(* IEC 61131-3 sources: programs/VI-54/VI-54_20171205/VI-54_20171205/Stations/Screen/LseClass170718/Class/TerminalControl, 1 file *)

(* ---- TerminalControl.st ---- *)
(*!
<Class
	Name               = "TerminalControl"
	Revision           = "3.2"
	RealtimeTask       = "false"
	CyclicTask         = "true"
	DefCyclictime      = "100 ms"
	BackgroundTask     = "false"
	Sigmatek           = "false"
	OSInterface        = "false"
	HighPriority       = "false"
	Automatic          = "false"
	UpdateMode         = "Prescan"
	SharedCommandTable = "true"
	Objectsize         = "(690,1560)">
	<Channels>
		<Server Name="ActScreenNbr" Visualized="true" Initialize="false" WriteProtected="true" Retentive="false"/>
		<Server Name="ActWindowNbr" Visualized="true" Initialize="false" WriteProtected="true" Retentive="false"/>
		<Server Name="Down" Visualized="true" Initialize="false" WriteProtected="true" Retentive="false"/>
		<Server Name="F1" Visualized="true" Initialize="false" WriteProtected="true" Retentive="false"/>
		<Server Name="F2" Visualized="true" Initialize="false" WriteProtected="true" Retentive="false"/>
		<Server Name="F3" Visualized="true" Initialize="false" WriteProtected="true" Retentive="false"/>
		<Server Name="F4" Visualized="true" Initialize="false" WriteProtected="true" Retentive="false"/>
		<Server Name="F5" Visualized="true" Initialize="false" WriteProtected="true" Retentive="false"/>
		<Server Name="F6" Visualized="true" Initialize="false" WriteProtected="true" Retentive="false"/>
		<Server Name="F7" Visualized="true" Initialize="false" WriteProtected="true" Retentive="false"/>
		<Server Name="F8" Visualized="true" Initialize="false" WriteProtected="true" Retentive="false"/>
		<Server Name="GoInReset" Visualized="true" Initialize="false" WriteProtected="false" Retentive="false"/>
		<Server Name="KeyCode" Visualized="true" Initialize="false" WriteProtected="true" Retentive="false"/>
		<Server Name="keypresCnt" Visualized="true" Initialize="false" WriteProtected="true" Retentive="false"/>
		<Server Name="Left" Visualized="true" Initialize="false" WriteProtected="true" Retentive="false"/>
		<Server Name="PgDown" Visualized="true" Initialize="false" WriteProtected="true" Retentive="false"/>
		<Server Name="PgUp" Visualized="true" Initialize="false" WriteProtected="true" Retentive="false"/>
		<Server Name="Right" Visualized="true" Initialize="false" WriteProtected="true" Retentive="false"/>
		<Server Name="sDeactivateScreenSaver" Visualized="true" Initialize="false" WriteProtected="false" Retentive="false"/>
		<Server Name="sDelayBacklight" Visualized="true" Initialize="true" WriteProtected="false" Retentive="File"/>
		<Server Name="sDelayScreenSaver" Visualized="true" Initialize="true" DefValue="0" WriteProtected="false" Retentive="File"/>
		<Server Name="SelectScreen" Visualized="true" Initialize="false" WriteProtected="false" Retentive="false"/>
		<Server Name="SelectWindow" Visualized="true" Initialize="false" WriteProtected="false" Retentive="false"/>
		<Server
			Name           = "Server0"
			Initialize     = "false"
			Visualized     = "true"
			WriteProtected = "true">
		</Server>
		<Server Name="Up" Visualized="true" Initialize="false" WriteProtected="true" Retentive="false"/>
		<Server Name="WindowEnd" Visualized="true" Initialize="false" WriteProtected="false" Retentive="false"/>
		<Client Name="OSkernel" Required="false" Internal="false"/>
	</Channels>
	<Network Name="TerminalControl">
		<!-- List of Components in this network -->
		<Components>
			<Object
				Name       = "_base"
				Class      = "_Global"
				Position   = "(270,150)"
				Visualized = "true">
				<Channels>
					<Server Name="Server0"/>
					<Client Name="Lse"/>
				</Channels>
			</Object>
		</Components>
		<Comments>
		</Comments>
		<!-- List of Connections in this network -->
		<Connections>
			<Connection Source="_base.Lse" Destination="this.Lse" Vertices="(270,240),(38,210),"/>
			<Connection Source="this.Server0" Destination="_base.Server0" Vertices="(742,210),(570,240),"/>
		</Connections>
		<!-- Headerfiles -->
		<Options>
		</Options>
	</Network>
</Class>
*)
#pragma using _Global

TerminalControl : CLASS
: _Global
  //Servers:
	SelectScreen 	: SvrCh_DINT;
	SelectWindow 	: SvrCh_DINT;
	ActWindowNbr 	: SvrCh_DINT;
	ActScreenNbr 	: SvrCh_DINT;
	KeyCode 	: SvrCh_DINT;
	keypresCnt 	: SvrCh_DINT;
	F1 	: SvrCh_DINT;
	F2 	: SvrCh_DINT;
	F3 	: SvrCh_DINT;
	F4 	: SvrCh_DINT;
	F5 	: SvrCh_DINT;
	F6 	: SvrCh_DINT;
	F7 	: SvrCh_DINT;
	F8 	: SvrCh_DINT;
	Up 	: SvrCh_DINT;
	Down 	: SvrCh_DINT;
	Left 	: SvrCh_DINT;
	Right 	: SvrCh_DINT;
	PgUp 	: SvrCh_DINT;
	PgDown 	: SvrCh_DINT;
	GoInReset 	: SvrCh_DINT;
	sDelayScreenSaver 	: SvrCh_UDINT;
	sDelayBacklight 	: SvrCh_UDINT;
	sDeactivateScreenSaver 	: SvrCh_DINT;
	WindowEnd 	: SvrCh_DINT;
  //Clients:
	OSkernel 	: CltChCmd__OSKernel;
  //Variables:
		LedF1Old 	: DINT;
		LedEROld 	: DINT;
		LedRNOld 	: DINT;
		LedF2Old 	: DINT;
		LedF3Old 	: DINT;
		LedF4Old 	: DINT;
		LedF5Old 	: DINT;
		LedF6Old 	: DINT;
		LedF7Old 	: DINT;
		LedF8Old 	: DINT;
		TimeMark 	: UDINT;
		dState_ScreenSaver 	: DINT;
		udTimeStamp 	: UDINT;
		ActScreenNbrOld 	: DINT;
		ActWindowNbrOld 	: DINT;
		Refresh 	: DINT;
  //Functions:

	FUNCTION VIRTUAL GLOBAL Init;

	FUNCTION VIRTUAL GLOBAL CyWork
		VAR_INPUT
			EAX 	: UDINT;
		END_VAR
		VAR_OUTPUT
			state (EAX) 	: UDINT;
		END_VAR;

	FUNCTION VIRTUAL GLOBAL IF_WindowRun
		VAR_INPUT
			whoami 	: ^_WHOAMI;
			pic 	: ^void;
			event 	: ^_EVENT;
		END_VAR;

	FUNCTION VIRTUAL GLOBAL IF_WindowEnd
		VAR_INPUT
			whoami 	: ^_WHOAMI;
			pic 	: ^void;
		END_VAR;
				//! <Function Comment="methode will be called after lse-project is successfully loaded and &#13;&#10;possibly given communication to extern plc is stable" Name="IF_ProjectReady"/>
	FUNCTION VIRTUAL GLOBAL IF_ProjectReady
		VAR_INPUT
			state 	: BOOL;
		END_VAR
		VAR_OUTPUT
			retcode 	: BOOL;
		END_VAR;

	FUNCTION GLOBAL SelectScreenNbr
		VAR_INPUT
			Nbr 	: DINT;
		END_VAR;

	FUNCTION GLOBAL SelectWindowNbr
		VAR_INPUT
			Nbr 	: DINT;
		END_VAR;

	FUNCTION GLOBAL ActScrnNbr
		VAR_OUTPUT
			ActNbr 	: DINT;
		END_VAR;

	FUNCTION GLOBAL ActWinNbr
		VAR_OUTPUT
			ActNbr 	: DINT;
		END_VAR;

	FUNCTION GLOBAL ResetScreen;

	FUNCTION VIRTUAL GLOBAL SelectScreen::Write
		VAR_INPUT
			input (EAX) 	: DINT;
		END_VAR
		VAR_OUTPUT
			result (EAX) 	: DINT;
		END_VAR;

	FUNCTION VIRTUAL GLOBAL SelectWindow::Write
		VAR_INPUT
			input (EAX) 	: DINT;
		END_VAR
		VAR_OUTPUT
			result (EAX) 	: DINT;
		END_VAR;

	FUNCTION VIRTUAL GLOBAL GoInReset::Write
		VAR_INPUT
			input (EAX) 	: DINT;
		END_VAR
		VAR_OUTPUT
			result (EAX) 	: DINT;
		END_VAR;

	FUNCTION VIRTUAL GLOBAL sDelayScreenSaver::Write
		VAR_INPUT
			input (EAX) 	: UDINT;
		END_VAR
		VAR_OUTPUT
			result (EAX) 	: UDINT;
		END_VAR;

	FUNCTION VIRTUAL GLOBAL sDelayBacklight::Write
		VAR_INPUT
			input (EAX) 	: UDINT;
		END_VAR
		VAR_OUTPUT
			result (EAX) 	: UDINT;
		END_VAR;
  //Tables:
	FUNCTION @STD
		VAR_OUTPUT
			ret_code	: CONFSTATES;
		END_VAR;
	FUNCTION GLOBAL TAB @CT_;
END_CLASS;

#pragma usingLtd _OSKernel

#pragma using _Lse

//*********************Inserted from .\MyGlobal\MyGlobal_00_00.st*********************

 //VIRTUAL GLOBAL MyGlobal::SelectScreen::Write

 //VIRTUAL GLOBAL MyGlobal::CyWork

FUNCTION VIRTUAL GLOBAL TerminalControl::IF_WindowRun
	VAR_INPUT
		whoami 	: ^_WHOAMI;
		pic 	: ^void;
		event 	: ^_EVENT;
	END_VAR

// check screen number..
	case whoami^.ima of

	IMA_PICTURE:
		ActScreenNbr := to_dint whoami^.no;

	IMA_WINDOW:
		ActWindowNbr := to_dint whoami^.no;
	end_case;

//  key control
	if event^.ftype = _event_keypress then
		KeyCode := event^.scancode;
  case event^.scancode of
			_F1: F1 := 1;
			_F2: F2 := 1;
			_F3: F3 := 1;
			_F4: F4 := 1;
			_F5: F5 := 1;
			_F6: F6 := 1;
			_F7: F7 := 1;
			_F8: F8 := 1;
			_UP: Up := 1;
			_DOWN : Down := 1;
			_LEFT : Left := 1;
			_RIGHT: Right := 1;
			_PGUP : PgUp := 1;
			_PGDOWN : PgDown := 1;
		end_case;
	elsif event^.ftype = _event_keyrelease then
		case event^.scancode of
			_F1:    F1 := 0;
			_F2:    F2 := 0;
			_F3:    F3 := 1;
			_F4:    F4 := 0;
			_F5:    F5 := 0;
			_F6:    F6 := 0;
			_F7:    F7 := 0;
			_F8:    F8 := 0;
			_UP:    Up := 0;
			_DOWN : Down := 0;
			_LEFT : Left := 0;
			_RIGHT: Right := 0;
			_PGUP : PgUp := 0;
			_PGDOWN : PgDown := 0;
		end_case;

		keypresCnt += 1;
	end_if;

  if (ActScreenNbr = 8 & SelectScreen = -1) then
    if ops.tAbsolute - TimeMark >= 30 * _100MS then
//      SelectScreen := 10;  not used !!
    end_if;
  else
    TimeMark := ops.tAbsolute;
  end_if;

// deactiveren van screen saver !!
  if ActScreenNbrOld <> ActScreenNbr then
    sDeactivateScreenSaver := 1;
  elsif ActWindowNbrOld <> ActWindowNbr then
    sDeactivateScreenSaver := 1;
  end_if;
  ActWindowNbrOld := ActWindowNbr;
  ActScreenNbrOld := ActScreenNbr;

// screen saver / backlight on/off
  if (whoami^.ima = IMA_SCREENSAVER) then
    case dState_ScreenSaver of

      0 : if sDelayBacklight > 0 then
            if ops.tAbsolute - udTimeStamp >= sDelayBacklight min then
              dState_ScreenSaver +=1;
            end_if;
          end_if;

    end_case;
    if sDeactivateScreenSaver <> 0 then
      // Deactivate the Screensaver and turns on the backlight
      sDeactivateScreenSaver :=0;
      reset_screensaver();
    end_if;
  else
    sDeactivateScreenSaver := 0;
  end_if;

END_FUNCTION //VIRTUAL GLOBAL MyGlobal::IF_WindowRun

FUNCTION VIRTUAL GLOBAL TerminalControl::IF_WindowEnd
	VAR_INPUT
		whoami 	: ^_WHOAMI;
		pic 	: ^void;
	END_VAR

	ActWindowNbr := 0;

END_FUNCTION

FUNCTION VIRTUAL GLOBAL TerminalControl::Init

// voer ook de oude init uit
	_Global::Init();
  SelectScreen := -1;
  SelectWindow := -1;

END_FUNCTION //VIRTUAL GLOBAL MyGlobal::Init

FUNCTION VIRTUAL GLOBAL TerminalControl::SelectScreen::Write
	VAR_INPUT
		input (EAX) 	: DINT;
	END_VAR
	VAR_OUTPUT
		result (EAX) 	: DINT;
	END_VAR

	SelectScreen := input;
 	result := SelectScreen;

END_FUNCTION

FUNCTION VIRTUAL GLOBAL TerminalControl::CyWork
	VAR_INPUT
		EAX 	: UDINT;
	END_VAR
	VAR_OUTPUT
		state (EAX) 	: UDINT;
	END_VAR

//                CMD_NEWPICTURE,     // open new picture (1)
//                CMD_NEWWINDOW,      // open new window (1)

	if SelectScreen <> - 1 then
    SelectScreenNbr(Nbr:=SelectScreen);
    SelectScreen := -1;
	end_if;

	if SelectWindow <> - 1 then
    SelectWindowNbr(Nbr:=SelectWindow);
    SelectWindow := -1;
	end_if;

   state:= READY;

END_FUNCTION

FUNCTION VIRTUAL GLOBAL TerminalControl::SelectWindow::Write
	VAR_INPUT
		input (EAX) 	: DINT;
	END_VAR
	VAR_OUTPUT
		result (EAX) 	: DINT;
	END_VAR

  InsertCmd(x0:=CMD_CLOSE, x1:= 0, x2:= 0);
	SelectWindow := input;
 	result := SelectWindow;

END_FUNCTION

FUNCTION GLOBAL TerminalControl::SelectScreenNbr
	VAR_INPUT
		Nbr 	: DINT;
	END_VAR

//                CMD_NEWPICTURE,     // open new picture (1)
//                CMD_NEWWINDOW,      // open new window (1)
		InsertCMD(CMD_NEWPICTURE, Nbr, 0);
			F1 := 0;  // bij scherm wissel Softkeys uitzetten
			F2 := 0;
			F3 := 1;
			F4 := 0;
			F5 := 0;
			F6 := 0;
			F7 := 0;
	    F8 := 0;
		  Up := 0;
      Down := 0;
	   	Left := 0;
			Right := 0;
			PgUp := 0;
			PgDown := 0;

END_FUNCTION

FUNCTION GLOBAL TerminalControl::SelectWindowNbr
	VAR_INPUT
		Nbr 	: DINT;
	END_VAR
//                CMD_NEWPICTURE,     // open new picture (1)
//                CMD_NEWWINDOW,      // open new window (1)

		InsertCMD(CMD_NEWWINDOW, Nbr, 0);
			F1 := 0;  // bij scherm wissel Softkeys uitzetten
			F2 := 0;
			F3 := 1;
			F4 := 0;
			F5 := 0;
			F6 := 0;
			F7 := 0;
	    F8 := 0;
		  Up := 0;
      Down := 0;
	   	Left := 0;
			Right := 0;
			PgUp := 0;
			PgDown := 0;

END_FUNCTION

FUNCTION GLOBAL TerminalControl::ActScrnNbr
	VAR_OUTPUT
		ActNbr 	: DINT;
	END_VAR

  ActNbr := ActScreenNbr;

END_FUNCTION

FUNCTION GLOBAL TerminalControl::ActWinNbr
	VAR_OUTPUT
		ActNbr 	: DINT;
	END_VAR

  ActNbr := ActWindowNbr;

END_FUNCTION

FUNCTION VIRTUAL GLOBAL TerminalControl::GoInReset::Write
	VAR_INPUT
		input (EAX) 	: DINT;
	END_VAR
	VAR_OUTPUT
		result (EAX) 	: DINT;
	END_VAR

	GoInReset := input;
  OSkernel.Reset();
 	result := GoInReset;

END_FUNCTION

FUNCTION GLOBAL TerminalControl::ResetScreen

    InsertCMD(CMD_NEWPICTURE, ActScreenNbr, 0);

END_FUNCTION

FUNCTION VIRTUAL GLOBAL TerminalControl::sDelayScreenSaver::Write
	VAR_INPUT
		input (EAX) 	: UDINT;
	END_VAR
	VAR_OUTPUT
		result (EAX) 	: UDINT;
	END_VAR

  // write the delay to the LSE kernel
	sDelayScreenSaver := input;  // in [min]
  Lse.DelayScreenSaver.Write(input := sDelayScreenSaver MIN);
 	result := sDelayScreenSaver;

END_FUNCTION

FUNCTION VIRTUAL GLOBAL TerminalControl::IF_ProjectReady
	VAR_INPUT
		state 	: BOOL;
	END_VAR
	VAR_OUTPUT
		retcode 	: BOOL;
	END_VAR

  // write delay to LSE kernel if the project is ready
  Lse.DelayScreenSaver.Write(input := sDelayScreenSaver min);
  retcode := state;

END_FUNCTION

FUNCTION VIRTUAL GLOBAL TerminalControl::sDelayBacklight::Write
	VAR_INPUT
		input (EAX) 	: UDINT;
	END_VAR
	VAR_OUTPUT
		result (EAX) 	: UDINT;
	END_VAR

	sDelayBacklight := input;
	result := sDelayBacklight;

END_FUNCTION
